{attribute 'GeneratedUsingTerminal: IODEVICETYPE_ETHERCATPROT'}
{attribute addProperty BoxType "IODEVICETYPE_ETHERCATPROT"}
{attribute addProperty Id "Beckhoff_EM2xxxBeckhoff_EM2xxx_C0B382EE40Beckhoff_EM3xxxBeckhoff_EM3xxx_3B040A8978Beckhoff_EM7xxxBeckhoff_EM7xxx_E01A06D1681SyncUnitsSyncUnits_99E584AF18InputsInputs_25A0042B160OutputsOutputs_2397A10E106InfoDataInfoData_E68C61CD28"}
{attribute addProperty CRC "4107517063"}
{attribute addProperty Size "1111"}
TYPE EtherCAT_Master_EMxxxx_F4D3BC87 :
STRUCT
	{attribute addProperty Name "Beckhoff_EM2xxx"}
	{attribute addProperty PreviousPort "EtherCAT_Master_EMxxxx : Master"}
	Beckhoff_EM2xxx : Beckhoff_EM2xxx_C0B382EE;
	{attribute addProperty Name "Beckhoff_EM3xxx"}
	{attribute addProperty PreviousPort "Beckhoff EM2xxx : C"}
	Beckhoff_EM3xxx : Beckhoff_EM3xxx_3B040A89;
	{attribute addProperty Name "Beckhoff_EM7xxx"}
	{attribute addProperty PreviousPort "Beckhoff EM3xxx : C"}
	Beckhoff_EM7xxx : Beckhoff_EM7xxx_E01A06D1;
	{attribute addProperty Name "SyncUnits"}
	SyncUnits : SyncUnits_99E584AF;
	{attribute addProperty Name "Inputs"}
	Inputs : Inputs_25A0042B;
	{attribute addProperty Name "Outputs"}
	Outputs : Outputs_2397A10E;
	{attribute addProperty Name "InfoData"}
	InfoData : InfoData_E68C61CD;
END_STRUCT
END_TYPE

(* stored: Version 1.2.0.0, ProductVersion 3.1.4024.9
   DUT EtherCAT_Master_EMxxxx_F4D3BC87: Id {16054cdd-0379-4804-b282-8fe026c19831} *)
